FUNCTION_BLOCK T_BoolCommandTask_1 EXTENDS T_MockCommandTask IMPLEMENTS I_BoolResultTask
VAR
  _result : BOOL;
END_VAR

PROPERTY Result : BOOL
GET
Result := _result;
END_GET
END_PROPERTY

METHOD PUBLIC SetResultValue
VAR_INPUT
  value : BOOL;
END_VAR
_result := value;
END_METHOD

END_FUNCTION_BLOCK

(* stored: Version 1.1.0.1
   POU T_BoolCommandTask_1: Id {ad74609e-ca9f-4daa-9bfd-ae4c36532e52}, SpecialFunc None
   Property Result: Id {c0e7327e-7e9b-4f8e-88e2-12ecb1dd9cdd}
   Get Get: Id {b182bdb7-242b-47ac-a801-e9455bf1a487}
   Method SetResultValue: Id {f417e13e-19ad-436b-954d-f2705314b636} *)
